{attribute 'GeneratedUsingTerminal: EJ2918-0000-0017'}
{attribute addProperty BoxType "EJ2918-0000-0017"}
{attribute addProperty Id "OutputsOutputs_FB9F35208"}
{attribute addProperty CRC "2551423886"}
{attribute addProperty Size "8"}
TYPE Module_2_FSOUT_9813A38E :
STRUCT
	{attribute addProperty Name "Outputs"}
	Outputs  : Outputs_FB9F3520;
END_STRUCT
END_TYPE

(* stored: Version 1.2.0.0, ProductVersion 3.1.4024.9
   DUT Module_2_FSOUT_9813A38E: Id {d0021624-9869-4229-843b-f1fa5e0e98f9} *)
